// Updates history curve
//
FUNCTION UpdateHistory: BOOL
VAR_INPUT
	
	Step: DINT; // Step counter (1...100)
	
END_VAR
VAR
	
	// Members...
	Index: INT; // Index of history point
	
END_VAR

//
IF Step <> 1 THEN

	RETURN;
	
END_IF

// Scan history data
FOR Index := NUM_HISTORY_POINTS TO 2 BY -1 DO

	//
	gstHistory.arPower[ Index ]       := gstHistory.arPower[ Index - 1 ];
	gstHistory.arTemperature[ Index ] := gstHistory.arTemperature[ Index - 1 ];
	gstHistory.arTempDiff[ Index ]    := gstHistory.arTemperature[ Index ] - gSetpoint;
	
END_FOR 

// Update newest data to history
gstHistory.arPower[ 1 ]       := LREAL_TO_REAL( gPower );
gstHistory.arTemperature[ 1 ] := IO_Inputs.i_HtrTemp;
gstHistory.arTempDiff[ 1 ]    := gstHistory.arTemperature[ 1 ] - gSetpoint;

END_FUNCTION

(* stored: Version 1.1.0.1, ProductVersion 3.1.4022.18
   POU UpdateHistory: Id {fa2b4187-9615-4f0d-9fed-4af5a48beba8}, SpecialFunc None *)
